// TIA Portal V19 export
TYPE "LEXCHANGETRAY_typeConstraintWorkstationIoSignalControlNode"
// reset: Bool
// monitoring: LEXCHANGETRAY_typeConstraintWorkstationIoSignalContronNodeMonitoring
// stored: Access Published
   STRUCT
      reset : Bool;
      monitoring { S7_SetPoint := 'True'} : "LEXCHANGETRAY_typeConstraintWorkstationIoSignalContronNodeMonitoring";
   END_STRUCT;
END_TYPE
